FUNCTION AboutEqual : BOOL
VAR_INPUT
	IN1: UINT;
	IN2: UINT;
	Tolerance: UINT;
END_VAR
VAR_OUTPUT
END_VAR
VAR
	Difference: UINT;
END_VAR

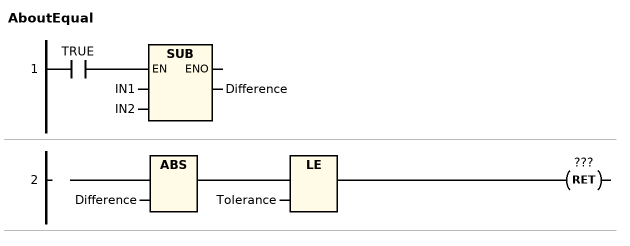
// NETWORK 1
Difference := IN1 - IN2;

// NETWORK 2
IF ABS(Difference) <= Tolerance THEN RETURN; END_IF

END_FUNCTION

(* stored: Version 1.1.0.1, ProductVersion 3.1.4024.12
   POU AboutEqual: Id {7f75b6ae-05cc-4911-8292-db1344cd16aa}, SpecialFunc None *)
